PROGRAM PRG_SERIAL_COM
VAR
END_VAR

(*Instanitate Serial port com function *) 
fbSerialLineControl(
	Mode:= SERIALLINEMODE_EL6_22B,
	pComIn:= ADR(stComIn),
	pComOut:=ADR(stComOut),
	SizeComIn:= SIZEOF(stComIn),
	TxBuffer:= SerialRXBuffer,
	RxBuffer:= SerialTXBuffer,
	Error=> ,
	ErrorID=> );

END_PROGRAM

(* stored: Version 1.1.0.1, ProductVersion 3.1.4020.14
   POU PRG_SERIAL_COM: Id {679ad23f-465a-4197-bd5e-90771d62ebf6}, SpecialFunc None *)
